// TwinCAT 3 PLC project Untitled1
// ProgramVersion: 3.1.4023.0
// libraries:
//   Tc2_Standard, * (Beckhoff Automation GmbH)
//   Tc2_System, * (Beckhoff Automation GmbH)
//   Tc3_Module, * (Beckhoff Automation GmbH)
// project tree:
//   FBs/Enumeration/ E_BoxPlaceDirection.TcDUT, E_RobotArmJointDirection.TcDUT
//   FBs/ FB_RobotArm.TcPOU
//   FBs/Structures/ ST_Inputs.TcDUT, ST_Outputs.TcDUT
//   GVLs/ GVL_RobotArm.TcGVL
//   / PlcTask.TcTTO
//   POUs/ MAIN.TcPOU
// real-time tasks:
//   TASK PlcTask: cycle T#10ms, priority 20, ADS port 350

CONFIGURATION Untitled1
    RESOURCE PLC ON TwinCAT3
        TASK PlcTask(INTERVAL := T#10ms, PRIORITY := 20);
        PROGRAM MAIN WITH PlcTask : MAIN;
    END_RESOURCE
END_CONFIGURATION

// ---- FBs/Enumeration/E_BoxPlaceDirection.TcDUT
{attribute 'qualified_only'}
{attribute 'strict'}
TYPE E_BoxPlaceDirection :
(
	PLACE1 := 1,
	PLACE2 := 2,
	PLACE3 := 3,
	
	LastPlace
);
END_TYPE

// ---- FBs/Enumeration/E_RobotArmJointDirection.TcDUT
{attribute 'qualified_only'}
{attribute 'strict'}
TYPE E_RobotArmJointDirection :
(
	RIGHT 	:= 1,
	LEFT	:= 2
);
END_TYPE

// ---- FBs/Structures/ST_Inputs.TcDUT
TYPE ST_Inputs :
STRUCT
	PLACE1            	: BOOL;
	PLACE2            	: BOOL;
	GRIP_CONDITION    	: BOOL;
	JOINT_RIGHT_SIGNAL	: ARRAY [1..4] OF BOOL;
	JOINT_LEFT_SIGNAL	: ARRAY [1..4] OF BOOL;
END_STRUCT
END_TYPE

// ---- FBs/Structures/ST_Outputs.TcDUT
TYPE ST_Outputs :
STRUCT
	GRIP_OPEN             : BOOL;
	GRIP_CLOSE            : BOOL;
	JOINT_TURN_LEFT   : ARRAY [1..4] OF BOOL;
	JOINT_TURN_RIGHT  : ARRAY [1..4] OF BOOL;
(*	JOINT_LEFT1_SIGNAL    : BOOL;
	JOINT_LEFT2_SIGNAL    : BOOL;
	JOINT_LEFT3_SIGNAL    : BOOL;
	JOINT_LEFT4_SIGNAL    : BOOL;
	JOINT_RIGHT1_SIGNAL   : BOOL;
	JOINT_RIGHT2_SIGNAL   : BOOL;
	JOINT_RIGHT3_SIGNAL   : BOOL;
	JOINT_RIGHT4_SIGNAL   : BOOL;  *)
END_STRUCT
END_TYPE

// ---- GVLs/GVL_RobotArm.TcGVL
{attribute 'qualified_only'}
VAR_GLOBAL CONSTANT
	NUMBER_OF_JOINTS : INT := 4;
END_VAR

// ---- POUs/MAIN.TcPOU
PROGRAM MAIN
VAR
	RobotArm			: FB_RobotArm;
//	RobotArm1Inputs 	: ST_Inputs;
//	RobotArm1Outputs 	: ST_Outputs;
	
//SerialIndex : INT:=1;
//Index : INT;


//LSTEPS   : INT;
//RSTEPS   : INT;

//START    : BOOL;
END_VAR

//RobotArm(ST_Inputs := RobotArm1Inputs, ST_Outputs := RobotArm1Outputs);

RobotArm();

END_PROGRAM

// ---- FBs/FB_RobotArm.TcPOU
FUNCTION_BLOCK FB_RobotArm
VAR
	Inputs 	AT%I* 	: ST_Inputs;
	Outputs AT%Q* 	: ST_Outputs;
	RobotArmJoints 	: ARRAY [1..GVL_RobotArm.NUMBER_OF_JOINTS] OF INT;
	Index 			: INT;
	
	//BoxPlaceLocation	: ARRAY [E_BoxPlaceDirection.PLACE1..E_BoxPlaceDirection.LastPlace] OF INT;
END_VAR

VAR PERSISTENT
	LSTEPS		: INT := 0;
	RSTEPS		: INT := 0;
	FirstScan 	: BOOL := TRUE;	
	
	InputsDecoupled		: ST_Inputs;
END_VAR

_M_StatusUpdate();


(*
	WRITE PUBLIC METHODS TO DO THE FOLLOWING:
	MOVE ONLY
		1. Move hand to Place #1
		2. Move hand to Place #2
		
	MOVE + GRIP
		3. PickUpFromPlace( placenum := x )
		4. PlaceTo( placenum := x )

*)

METHOD PRIVATE _M_DefaultPosition : BOOL
VAR
	Index		: INT;
END_VAR
_M_GripControl( Close := TRUE ); // METHOD( INPUT := , OUTPUT => )
	
FOR Index := 1 TO GVL_RobotArm.NUMBER_OF_JOINTS DO 
	Outputs.JOINT_TURN_LEFT[Index] := FALSE;
	Outputs.JOINT_TURN_RIGHT[Index]:=FALSE;//optimisation of//inputs.JOINT_TURN_RIGHT1:=inputs.JOINT_TURN_RIGHT2:=inputs.JOINT_TURN_RIGHT3:=inputs.JOINT_TURN_RIGHT4:=FALSE;
		
	LSTEPS:=RSTEPS:=0; // Will it be understandable?
END_FOR
END_METHOD

METHOD PRIVATE _M_GripControl : BOOL
VAR_INPUT
	Close	: BOOL;
END_VAR
Outputs.GRIP_CLOSE := Close;
Outputs.GRIP_OPEN := NOT Close;
END_METHOD

METHOD PRIVATE _M_StatusUpdate : BOOL
VAR_INPUT
END_VAR
InputsDecoupled.GRIP_CONDITION := Inputs.GRIP_CONDITION;
END_METHOD

METHOD PRIVATE _M_StraightJoint : BOOL
VAR
	Joint				: INT :=1;
END_VAR
Outputs.GRIP_CLOSE:=TRUE;

Outputs.JOINT_TURN_LEFT[Joint] := FALSE;
Outputs.JOINT_TURN_RIGHT[Joint] := FALSE;

//FOR Index := 1 TO GVL_RobotArm.NUMBER_OF_JOINTS BY 1 DO
//	inputs.JOINT_TURN_LEFT[Index]:=FALSE;
//	inputs.JOINT_TURN_RIGHT[Index]:=FALSE;
//END_FOR

(* CASE StraightPosition OF 
1:	inputs.JOINT_TURN_LEFT1:=FALSE;
	inputs.JOINT_TURN_RIGHT1:=FALSE;
2: 	inputs.JOINT_TURN_LEFT2:=FALSE;
	inputs.JOINT_TURN_RIGHT2:=FALSE;
3: 	inputs.JOINT_TURN_LEFT3:=FALSE;
	inputs.JOINT_TURN_RIGHT3:=FALSE;
4: 	inputs.JOINT_TURN_LEFT4:=FALSE;
	inputs.JOINT_TURN_RIGHT4:=FALSE;	
END_CASE *)
END_METHOD

METHOD PUBLIC M_PickUpFromPlace : BOOL
VAR_INPUT
	PLACE_NUM : INT;
END_VAR
(*

	1. Return to default position 
	2. Move hand to Place 1
	3. Open Grip
	4. Close Grip when picked up (picked up => GRIP_CONDITION = TRUE)
	...
	optionally: return to default position

*)
_M_DefaultPosition();

M_TurnJoint( TurnDirection := E_RobotArmJointDirection.LEFT, Joint := 2);


IF outputs.GRIP_OPEN THEN
	outputs.GRIP_CLOSE		:=FALSE;
	inputs.PLACE1			:=TRUE;
	inputs.GRIP_CONDITION	:=FALSE;
ELSIF inputs.GRIP_CONDITION THEN
	Outputs.GRIP_CLOSE		:=TRUE;
	_M_DefaultPosition();
END_IF
END_METHOD

METHOD PUBLIC M_Place1 : BOOL
VAR_INPUT
END_VAR

(*

	1. Return to default position 
	2. Move hand to Place 1
	3. Open Grip 
	...
	optionally: return to default position BUT returning to default must be performed ONLY IF GRIP_CONDITION EMPTY

*)
_M_DefaultPosition(Default:=TRUE);
M_TurnJoint(TurnDirection:='LEFT');
outputs.GRIP_OPEN:=FALSE;

IF Inputs.GRIP_CONDITION THEN
	inputs.GRIP_CONDITION:=FALSE;
 _M_DefaultPosition(Default:=TRUE);

END_IF
END_METHOD

METHOD PUBLIC M_Place2 : BOOL
VAR_INPUT
END_VAR
(*

	1. Return to default position 
	2. Move hand to Place 2
	3. Open Grip
	...
	optionally: return to default position BUT returning to default must be performed ONLY IF GRIP_CONDITION EMPTY

*)

_M_DefaultPosition(Default:=TRUE);
M_TurnJoint(TurnDirection:='RIGHT');
outputs.GRIP_OPEN:=TRUE;

IF outputs.GRIP_OPEN THEN
	inputs.GRIP_CONDITION:=FALSE;
 _M_DefaultPosition(Default:=TRUE);

END_IF
END_METHOD

METHOD PUBLIC M_PlaceTo : BOOL
VAR_INPUT
	PLACE_NUM : INT;
END_VAR
(*

	1. Return to default position 
	2. Move hand to Place 2
	3. Open Grip
	4. Close Grip when picked up (picked up => GRIP_CONDITION = TRUE)
	...
	optionally: return to default position

*)
_M_DefaultPosition(Default:=TRUE);
M_TurnJoint(TurnDirection:='RIGHT');
IF inputs.GRIP_CONDITION THEN
	outputs.GRIP_OPEN		:=TRUE;
	inputs.PLACE2			:=FALSE;
ELSIF inputs.GRIP_CONDITION:=FALSE THEN
	_M_DefaultPosition(Default:=TRUE);
END_IF
END_METHOD

METHOD PUBLIC M_TurnJoint : BOOL
VAR_INPUT
	TurnDirection 	: INT;
	Joint			: INT;
END_VAR
CASE TurnDirection OF 
	E_RobotArmJointDirection.LEFT: // turn left
		Outputs.JOINT_TURN_LEFT[Joint] := TRUE;
	E_RobotArmJointDirection.RIGHT: // turn right
		Outputs.JOINT_TURN_RIGHT[Joint] := TRUE;
END_CASE
END_METHOD

END_FUNCTION_BLOCK
